(* CODESYS project Portal Simple Example Process.project

Project tree, tasks and I/O mapping:
  Device : CODESYS Control for Raspberry Pi, 3S - Smart Software Solutions GmbH, version 3.5.11.20
    application Application
      libraries: Standard, * (System); Util, * (System); VisuDialogs, * (System)
      task MainTask (cyclic, interval 4 ms, priority 1) calls PLC_PRG
      task Profinet_IOTask (cyclic, interval t#1ms, priority 1) calls nothing
      task Profinet_CommunicationTask (cyclic, interval t#10ms, priority 30) calls PN_Controller.CommCycle
      task VISU_TASK (cyclic, interval 100 ms, priority 31) calls VisuElems.Visu_Prg
      program PLC_PRG [CFC]
      data type Position
      data type TwoByteOverInteger
      function block EinfachePortalsteuerung [ST]
      visualisation Visualization
      function block AnimationSteuerung [ST]
    SoftMotion General Axis Pool
    I²C
    SPI
    GPIOs_A_B : GPIOs A/B, 3S - Smart Software Solutions GmbH, version 3.5.11.0
        unmapped channels: digital inputs (GPIO0..GPIO31), digital outputs (GPIO0..GPIO31)
    Onewire
    Camera device
      <Leer>
    Ethernet : Ethernet, 3S - Smart Software Solutions GmbH, version 3.5.11.0
        settings: IPAddress = [192,168,176,1]; SubnetMask = [255,255,255,0]; GatewayAddress = [0,0,0,0]; MACAddress = [16#F4,16#F2,16#6D,16#18,16#1A,16#67]; NetworkInterfaceName = 'eth1'; NetworkInterfaceName = "eth1"; SaveCommunicationSettings = FALSE
      PN_Controller : PN-Controller, 3S - Smart Software Solutions GmbH, order no. 1, version 3.5.11.30
          settings: First IP Address = [192, 168, 176, 78]; Last IP Address = [192, 168, 176, 80]; Default Subnet Mask = [255, 255, 255, 0]; Default Gateway Address = [0, 0, 0, 0]; PDPortDataCheck.PeerStationName = ''
        Portal : Portal, BBS Brinkstraße, order no. 6ES7 214-1AG40-0XB0, version SW=V4.2, HW=
            settings: Slave parameters.Identification.IP address = [192,168,176,78]; Slave parameters.Identification.Subnet mask = [255,255,255,0]; Slave parameters.Identification.Default gateway = [0,0,0,0]; Slave parameters.Identification.MAC address = [16#00,16#00,16#00,16#00,16#00,16#00]; Slave parameters.Identification.Station name = 'portal6'; Slave parameters.Reduction ratio = 16; Slave parameters.Watchdog interval = 15; swapInfoOutputs = [10,6,7,5,10,1,2,15]; swapInfoInputs = [10,6,7,5,2,16]; swapInfoOutputs = [10,2,2,126]; swapInfoInputs = [10,2,2,126]; PDPortDataCheck.PeerStationName = ''
            output Application.PLC_PRG.LedStart : BOOL  // Outputs.Portal In Panel.LED Start
            output Application.PLC_PRG.LedReset : BOOL  // Outputs.Portal In Panel.LED Reset
            output Application.PLC_PRG.MotorenAktivieren : BOOL  // Outputs.Portal In Control.Motoren einschalten
            output Application.PLC_PRG.GreiferOeffnen : BOOL  // Outputs.Portal In Control.Greifer öffnen
            output Application.PLC_PRG.GreiferSchliessen : BOOL  // Outputs.Portal In Control.Greifer schließen
            output Application.PLC_PRG.StartHoming : BOOL  // Outputs.Portal In Move.Referenzfahrt starten
            output Application.PLC_PRG.StartPositionierungXY : BOOL  // Outputs.Portal In Move.Positionierung XY starten
            output Application.PLC_PRG.StartPositionierungZ : BOOL  // Outputs.Portal In Move.Positionierung Z starten
            output Application.PLC_PRG.SollPositionX : INT  // Outputs.Position X (0,1 mm)
            output Application.PLC_PRG.SollPositionY : INT  // Outputs.Position Y (0,1 mm)
            output Application.PLC_PRG.SollPositionZ : INT  // Outputs.Position Z (0,1 mm)
            input  Application.PLC_PRG.StartButton : BOOL  // Inputs.Portal Out Panel.Button Start
            input  Application.PLC_PRG.StopButton : BOOL  // Inputs.Portal Out Panel.Button Stop
            input  Application.PLC_PRG.ResetButton : BOOL  // Inputs.Portal Out Panel.Button Reset
            input  Application.PLC_PRG.MotorenAktiv : BOOL  // Inputs.Portal Out Control State.Motoren eingeschaltet
            input  Application.PLC_PRG.GreiferAuf : BOOL  // Inputs.Portal Out Control State.Greifer offen
            input  Application.PLC_PRG.GreiferZu : BOOL  // Inputs.Portal Out Control State.Greifer geschlossen
            input  Application.PLC_PRG.HomingFertig : BOOL  // Inputs.Portal Out Move State.Referenzfahrt fertig
            input  Application.PLC_PRG.PositionXYFertig : BOOL  // Inputs.Portal Out Move State.Positionierung XY fertig
            input  Application.PLC_PRG.PositionZFertig : BOOL  // Inputs.Portal Out Move State.Positionierung Z fertig
            input  Application.PLC_PRG.IstPositionX : INT  // Inputs.Position X (0,1 mm)
            input  Application.PLC_PRG.IstPositionY : INT  // Inputs.Position Y (0,1 mm)
            input  Application.PLC_PRG.IstPositionZ : INT  // Inputs.Position Z (0,1 mm)
            output Application.PLC_PRG.LesenStarten : BOOL  // Outputs.Rfid In Control.Lesen starten
            output Application.PLC_PRG.SchreibenStarten : BOOL  // Outputs.Rfid In Control.Schreiben starten
            output Application.PLC_PRG.SchreibDaten  // Outputs.RfidIn
            input  Application.PLC_PRG.TagVorhanden : BOOL  // Inputs.Rfid Out Control.Tag vorhanden
            input  Application.PLC_PRG.RfidFertig : BOOL  // Inputs.Rfid Out Control.RFID fertig
            input  Application.PLC_PRG.LeseDaten  // Inputs.RfidOut
            unmapped channels: Outputs, Inputs, Outputs, Inputs
  text list GlobalTextList
*)

// Device/Application/Position
TYPE Position :
STRUCT
	X: INT;
	Y: INT;
	Z: INT;
END_STRUCT
END_TYPE

// Device/Application/TwoByteOverInteger
TYPE TwoByteOverInteger :
UNION
	i: INT;
	bytes: ARRAY [0..1] OF BYTE;
END_UNION
END_TYPE

// Device/Application/PLC_PRG
PROGRAM PLC_PRG
VAR
	Portal1: EinfachePortalsteuerung;
	GreiferZu: BOOL;
	GreiferAuf: BOOL;
	GreiferSchliessen: BOOL;
	GreiferOeffnen: BOOL;
	AnimationSteuerung_0: AnimationSteuerung;
	MotorenAktiv: BOOL;
	HomingFertig: BOOL;
	PositionZFertig: BOOL;
	PositionXYFertig: BOOL;
	IstPositionX: INT;
	IstPositionY: INT;
	IstPositionZ: INT;
	MotorenAktivieren: BOOL;
	StartHoming: BOOL;
	SollPositionX: INT;
	SollPositionY: INT;
	SollPositionZ: INT;
	StartPositionierungZ: BOOL;
	StartPositionierungXY: BOOL;
	StartButton: BOOL;
	StopButton: BOOL;
	ResetButton: BOOL;
	LedStart: BOOL;
	LedReset: BOOL;
	LeseDaten: ARRAY [0..125] OF BYTE;
	SchreibDaten: ARRAY [0..125] OF BYTE;
	TagVorhanden: BOOL;
	RfidFertig: BOOL;
	StarteLesen: BOOL;
	StarteSchreiben: BOOL;
	LesenStarten: BOOL;
	SchreibenStarten: BOOL;
END_VAR

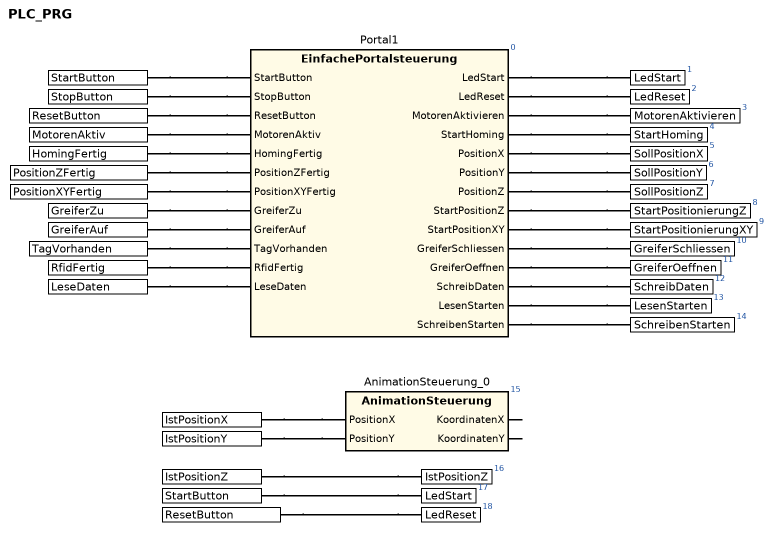
// note: 5 stored wires end on pins the file does not list and are not shown
Portal1(
    StartButton := StartButton,
    StopButton := StopButton,
    ResetButton := ResetButton,
    MotorenAktiv := MotorenAktiv,
    HomingFertig := HomingFertig,
    PositionZFertig := PositionZFertig,
    PositionXYFertig := PositionXYFertig,
    GreiferZu := GreiferZu,
    GreiferAuf := GreiferAuf,
    TagVorhanden := TagVorhanden,
    RfidFertig := RfidFertig,
    LeseDaten := LeseDaten); // EinfachePortalsteuerung
LedStart := Portal1.LedStart;
LedReset := Portal1.LedReset;
MotorenAktivieren := Portal1.MotorenAktivieren;
StartHoming := Portal1.StartHoming;
SollPositionX := Portal1.PositionX;
SollPositionY := Portal1.PositionY;
SollPositionZ := Portal1.PositionZ;
StartPositionierungZ := Portal1.StartPositionZ;
StartPositionierungXY := Portal1.StartPositionXY;
GreiferSchliessen := Portal1.GreiferSchliessen;
GreiferOeffnen := Portal1.GreiferOeffnen;
SchreibDaten := Portal1.SchreibDaten;
LesenStarten := Portal1.LesenStarten;
SchreibenStarten := Portal1.SchreibenStarten;
AnimationSteuerung_0(PositionX := IstPositionX, PositionY := IstPositionY); // AnimationSteuerung
IstPositionZ := IstPositionZ;
LedStart := StartButton;
LedReset := ResetButton;

END_PROGRAM

// Device/Application/EinfachePortalsteuerung
FUNCTION_BLOCK EinfachePortalsteuerung
VAR_INPUT
	// Buttons
	StartButton: BOOL;
	StopButton: BOOL;
	ResetButton: BOOL;
	// Portal
	MotorenAktiv: BOOL;
	HomingFertig: BOOL;
	PositionZFertig: BOOL;
	PositionXYFertig: BOOL;
	// Greifer
	GreiferZu: BOOL;
	GreiferAuf: BOOL;
	// RFID
	TagVorhanden: BOOL;
	RfidFertig: BOOL;
	LeseDaten: ARRAY [0..125] OF BYTE;
END_VAR
VAR_OUTPUT
	// Buttons
	LedStart: BOOL;
	LedReset: BOOL;
	// Portal
	MotorenAktivieren: BOOL;
	StartHoming: BOOL;
	PositionX: INT;
	PositionY: INT;
	PositionZ: INT;
	StartPositionZ: BOOL;
	StartPositionXY: BOOL;
	// Greifer
	GreiferSchliessen: BOOL;
	GreiferOeffnen: BOOL;
	// RFID
	SchreibDaten: ARRAY [0..125] OF BYTE;
	LesenStarten: BOOL;
	SchreibenStarten: BOOL;
END_VAR
VAR
	iStep: INT;
	Produktaufnahme: Position;
	Produktablage: Position;
	RfidPosition: Position;
	SchieberGreifposition: Position;
	delay: TON;
	blinker: Blink;
	Fahrthoehe: INT;
END_VAR


// wichtige Koordinaten
Produktaufnahme.X := 500; 
Produktaufnahme.Y := 3000; 
Produktaufnahme.Z := 10;

Produktablage.X := 3900; 
Produktablage.Y := 3000; 
Produktablage.Z := 10;

RfidPosition.X := 2000; 
RfidPosition.Y := 3700; 
RfidPosition.Z := 470;

SchieberGreifposition.X := 2000; 
SchieberGreifposition.Y := 3000; 
SchieberGreifposition.Z := 110;

Fahrthoehe := 460;


// LED in Tastern blinken lassen
blinker(enable:=TRUE, timehigh:=T#0.5S, timelow:=T#0.5S);
LedStart := (iStep > 100) OR (iStep = 100 AND blinker.OUT);
LedReset := (iStep = 30) OR (iStep = 10 AND blinker.OUT);

IF NOT StopButton THEN
    iStep := 0;
END_IF;

// Schrittkette abarbeiten
CASE iStep OF

	0:
        iStep := 10;
		
        // ######## Grundstellung anfahren ###########   

    10:
		delay(IN := FALSE, PT := T#10S);
        IF ResetButton THEN 
            MotorenAktivieren := TRUE;
            iStep := 20;
        END_IF;

    20:
        IF MotorenAktiv THEN
            StartHoming := TRUE;
            iStep := 30;
        END_IF;

    30:
        IF HomingFertig THEN
            StartHoming := FALSE;
            iStep := 40;
        END_IF;
		
	40:
		GreiferOeffnen := TRUE;
		IF GreiferAuf THEN	
			GreiferOeffnen := FALSE;
            iStep := 100;
        END_IF;	

        // ######## Start der Automatik ###########   
		
	100:
	    // Fahre zur Produktaufnahme, erst wenn Starttaster gedrückt wird
        IF StartButton THEN
            iStep := 105;
        END_IF;
	
	105:
		delay(IN := TRUE, PT := T#10S);
		IF delay.Q THEN
			delay(IN := FALSE, PT := T#10S);
			iStep := 110;
		END_IF;

	110:
		// Starte Fahrt in XY-Richtung
		PositionX := Produktaufnahme.X;
		PositionY := Produktaufnahme.Y;
		StartPositionXY := TRUE;
		IF PositionXYFertig THEN
			StartPositionXY := FALSE;
			iStep := 120;
		END_IF;
			
    120:
		// Starte Fahrt in Z-Richtung
		PositionZ := Produktaufnahme.Z;
        StartPositionZ := TRUE;
		IF PositionZFertig THEN	
        	StartPositionZ := FALSE;
			iStep := 130;
		END_IF;

	130:
		// Schließe Greifer, wenn in Aufnahmeposition
		GreiferSchliessen := TRUE;
		IF  GreiferZu THEN	
			GreiferSchliessen := FALSE;
            iStep := 140;
        END_IF;	

    140:
		// Fahrt in Z-Richtung nach oben
		PositionZ := Fahrthoehe;
		StartPositionZ := TRUE;
		IF PositionZFertig THEN	
        	StartPositionZ := FALSE;
			iStep := 150;
		END_IF;	

    150:
	    // Starte Fahrt in XY-Richtung zum RFID-Leser
		PositionX := RfidPosition.X;
        PositionY := RfidPosition.Y;
        StartPositionXY := TRUE;
        IF PositionXYFertig THEN
            StartPositionXY := FALSE;
            iStep := 160;
        END_IF;

    160:
		// warte auf RFID-Tag
		IF TagVorhanden THEN
			iStep := 170;
        END_IF;
		
	170:
		// lese RFID von Produkt
		LesenStarten := TRUE;
		IF RfidFertig THEN
			LesenStarten := FALSE;
			iStep := 180;
		END_IF;
		
	180:
		// Starte Fahrt in XY-Richtung zur Ablage
		PositionX := Produktablage.X;
        PositionY := Produktablage.Y;
        StartPositionXY := TRUE;
        IF PositionXYFertig THEN
            StartPositionXY := FALSE;
            iStep := 190;
        END_IF;
		
	190:
		// Fahrt in Z-Richtung zur Ablage
		PositionZ := Produktablage.Z;
		StartPositionZ := TRUE;
		IF PositionZFertig THEN	
        	StartPositionZ := FALSE;
			iStep := 200;
		END_IF;	
		
	200:
		// Öffne Greifer, wenn in Ablageposition
		GreiferOeffnen := TRUE;
		IF  GreiferAuf THEN	
			GreiferOeffnen := FALSE;
            iStep := 210;
        END_IF;	
		
	210:
		// Fahrt in Z-Richtung auf volle Höhe
		PositionZ := Fahrthoehe;
		StartPositionZ := TRUE;
		IF PositionZFertig THEN	
        	StartPositionZ := FALSE;
			iStep := 220;
		END_IF;	

	220:
		// Starte Fahrt in XY-Richtung zum Schieber
		PositionX := SchieberGreifposition.X;
        PositionY := SchieberGreifposition.Y;
        StartPositionXY := TRUE;
        IF PositionXYFertig THEN
            StartPositionXY := FALSE;
            iStep := 230;
        END_IF;
		
	230:
		// Fahrt in Z-Richtung zum Schieber
		PositionZ := SchieberGreifposition.Z;
		StartPositionZ := TRUE;
		IF PositionZFertig THEN	
        	StartPositionZ := FALSE;
			iStep := 240;
		END_IF;	
		
	240:
		// Schiebe Produkt aus Maschine
		PositionX := SchieberGreifposition.X + 500;
        PositionY := SchieberGreifposition.Y;
        StartPositionXY := TRUE;
        IF PositionXYFertig THEN
            StartPositionXY := FALSE;
            iStep := 250;
        END_IF;
	
	250:
		// Schiebe Schieber zurück an Ausgangsposition
		PositionX := SchieberGreifposition.X;
        PositionY := SchieberGreifposition.Y;
        StartPositionXY := TRUE;
        IF PositionXYFertig THEN
            StartPositionXY := FALSE;
            iStep := 260;
        END_IF;
		
	260:
		// Fahrt in Z-Richtung zurück auf volle Höhe
		PositionZ := Fahrthoehe;
		StartPositionZ := TRUE;
		IF PositionZFertig THEN	
        	StartPositionZ := FALSE;
			iStep := 300;
		END_IF;

	300:
		delay(IN := TRUE, PT := T#5S);
		IF delay.Q THEN
			delay(IN := FALSE, PT := T#5S);
			iStep := 0;
		END_IF;

END_CASE;

END_FUNCTION_BLOCK

// Device/Application/AnimationSteuerung
FUNCTION_BLOCK AnimationSteuerung
VAR_INPUT
	PositionX: INT;
	PositionY: INT;
END_VAR
VAR_OUTPUT
	KoordinatenX: INT;
	KoordinatenY: INT;
END_VAR
VAR
END_VAR


KoordinatenX := (PositionX / 10);
KoordinatenY := 390 - (PositionY / 10);

END_FUNCTION_BLOCK

// Device/Application/Visualization
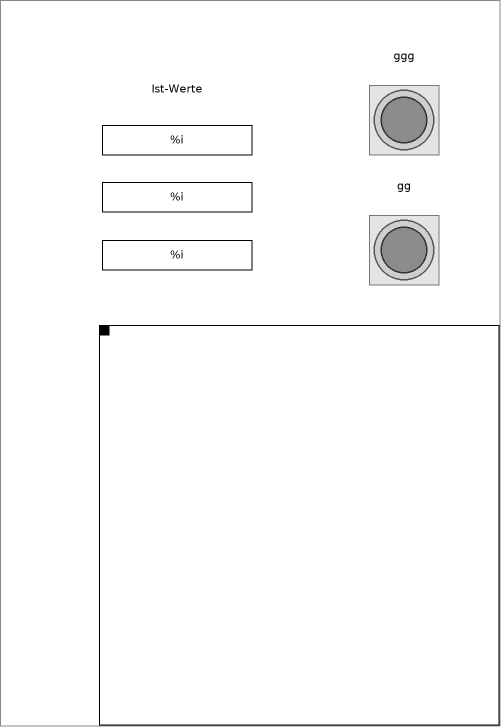
VISUALIZATION Visualization  // 501x727
    Rectangle (102,125 150x30), "%i", text variable: PLC_PRG.IstPositionX
    Rectangle (102,182 150x30), "%i", text variable: PLC_PRG.IstPositionY
    Rectangle (102,240 150x30), "%i", text variable: PLC_PRG.IstPositionZ
    Rectangle (102,74 150x30), "Ist-Werte"
    PushSwitch (369,85 70x70), behaviour: TAP, style: Switch-PushSwitch-Gray
    Rectangle (329,41 150x30), "ggg"
    PushSwitch (369,215 70x70), behaviour: TAP, style: Switch-PushSwitch-Gray
    Rectangle (329,171 150x30), "gg"
    Rectangle (99,325 400x400)
    Rectangle (99,325 10x10)
        p874137650: PLC_PRG.AnimationSteuerung_0.KoordinatenX
        p1126004900: PLC_PRG.AnimationSteuerung_0.KoordinatenY
        p3528305787: PLC_PRG.AnimationSteuerung_0.KoordinatenX
        p2773130477: PLC_PRG.AnimationSteuerung_0.KoordinatenY
END_VISUALIZATION
